// TIA Portal V19 export
DATA_BLOCK "A02_TrkManager"   // DB2534
// stored: InstanceOfName A02_TrkManager_FB, InstanceOfType FB
"A02_TrkManager_FB"
   // VAR_INPUT
   //    AreaInterface : "AreaInterface";
   //    SuperUserLogged : Bool;
   // END_VAR
   // VAR
   //    HMI : Struct
   //       A0202 : Struct
   //          Move : Array[1.."PTRK_A0202_ITEMS"] of "TrkMng_Move";
   //          NumDelete { S7_SetPoint := 'True'} : Int;
   //       END_STRUCT;
   //       A020_EXIT : Struct
   //          ButtonRecondVisibility : Array[1.."PTRK_A0202_EXIT_TOCHECK_ITEMS"] of Bool;
   //       END_STRUCT;
   //    END_STRUCT;
   //    Sts : Struct
   //       MoveA0202 : Struct
   //          SelectionOn : Bool;
   //          SelectionNo : Int;
   //       END_STRUCT;
   //    END_STRUCT;
   //    A0202_TON_Delete_Buttons : IEC_TIMER;
   // END_VAR
BEGIN
END_DATA_BLOCK
